SUBAPPLICATION SS1 (* Subapplication Type *)
  (* Standard: 61499-2 *)
  (* Version 1.0, 2024-07-25, DEVIASH *)
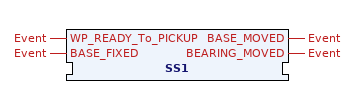
  EVENT_INPUT
    WP_READY_To_PICKUP; (* Initialization Request *)
    BASE_FIXED;
  END_EVENT
  EVENT_OUTPUT
    BASE_MOVED; (* Initialization Confirm *)
    BEARING_MOVED;
  END_EVENT
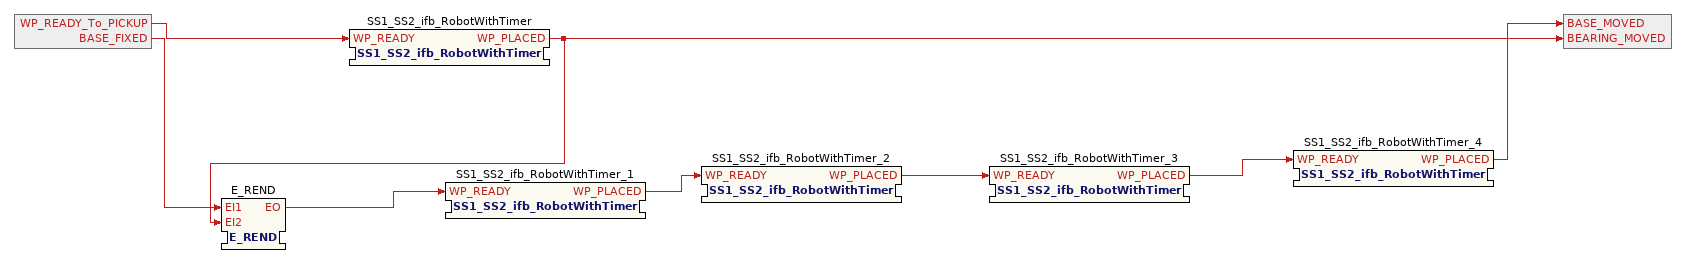
  FBS
    E_REND : E_REND;
    SS1_SS2_ifb_RobotWithTimer : SS1_SS2_ifb_RobotWithTimer;
    SS1_SS2_ifb_RobotWithTimer_1 : SS1_SS2_ifb_RobotWithTimer;
    SS1_SS2_ifb_RobotWithTimer_2 : SS1_SS2_ifb_RobotWithTimer;
    SS1_SS2_ifb_RobotWithTimer_3 : SS1_SS2_ifb_RobotWithTimer;
    SS1_SS2_ifb_RobotWithTimer_4 : SS1_SS2_ifb_RobotWithTimer;
  END_FBS
  EVENT_CONNECTIONS
    WP_READY_To_PICKUP TO SS1_SS2_ifb_RobotWithTimer.WP_READY;
    SS1_SS2_ifb_RobotWithTimer_1.WP_PLACED TO SS1_SS2_ifb_RobotWithTimer_2.WP_READY;
    SS1_SS2_ifb_RobotWithTimer_2.WP_PLACED TO SS1_SS2_ifb_RobotWithTimer_3.WP_READY;
    SS1_SS2_ifb_RobotWithTimer_3.WP_PLACED TO SS1_SS2_ifb_RobotWithTimer_4.WP_READY;
    BASE_FIXED TO E_REND.EI1;
    SS1_SS2_ifb_RobotWithTimer.WP_PLACED TO E_REND.EI2;
    E_REND.EO TO SS1_SS2_ifb_RobotWithTimer_1.WP_READY;
    SS1_SS2_ifb_RobotWithTimer_4.WP_PLACED TO BASE_MOVED;
    SS1_SS2_ifb_RobotWithTimer.WP_PLACED TO BEARING_MOVED;
  END_CONNECTIONS
END_SUBAPPLICATION
